PROGRAM MAIN
VAR
END_VAR

P_ScaleSensors();
P_out();
P_VHMI();
P_ControlSystem();

END_PROGRAM

(* stored: Version 1.1.0.1, ProductVersion 3.1.4024.12
   POU MAIN: Id {99aa5d7f-5074-4316-ab0f-83e396c2057c}, SpecialFunc None *)
